// TIA Portal V20 export
TYPE "LER_typeRFIDMonitoring"
// stored: Access Published
   STRUCT
      ResultData : "LSicar_typeIdentInterfaceHmi";
      error : Bool;
      status : DWord;
   END_STRUCT;
END_TYPE
